// TIA Portal V16 export
// export: Created 2023-03-29T11:03:22.7150426Z, ExportSetting WithDefaults, DisplayName Totally Integrated Automation Portal, DisplayVersion V16 Update 6, DisplayName TIA Portal Version Control Interface, DisplayVersion V16 Update 2, DisplayName TIA Portal Openness, DisplayVersion V16 Update 6, DisplayName STEP 7 Professional, DisplayVersion V16 Update 6, DisplayName STEP 7 Safety, DisplayVersion V16, DisplayName WinCC Advanced, DisplayVersion V16 Update 6
FUNCTION_BLOCK "Startegia_sterowania"   // FB18, LAD
TITLE = Strategia przełączania
{ S7_Optimized_Access := 'TRUE' }
AUTHOR : rtecmer
VERSION : 0.1
// Funkcja przełącza stan aktywnego zbiornika w trybie napełniania i opróróżniana. Cykl pracy . Zbiornik opróżniany zostaje aktywny do napełniania a jeden pełny aktywny do przetłaczannia. 
// Znacznik blok_tank_x - blukuje zbiornik po zakonczonym cyklu do czasu aż wszystkie zbiorniki nie przejdą sekwencji.
// stored: AutoNumber true, IsIECCheckEnabled false, IsRetainMemResEnabled false, MemoryReserve 250, SetENOAutomatically false, UDAEnableTagReadback false
   VAR
      tmp_time_1 : Bool;   // pomocniczy bit do wyzwolenia opóźnionego resetu aktywnego zbiornika
      tmp_time_2 : Bool := false;   // pomocniczy bit do wyzwolenia opóźnionego resetu aktywnego zbiornika
      tmp_time_3 : Bool := false;   // pomocniczy bit do wyzwolenia opóźnionego resetu aktywnego zbiornika
      tmp_time_4 : Bool := false;   // pomocniczy bit do wyzwolenia opóźnionego resetu aktywnego zbiornika
   END_VAR
   VAR_TEMP   // added for the SCL form of the ladder/FBD networks
      _w1 : Bool;
      _w2 : Bool;
   END_VAR
BEGIN

REGION Network 2: jest zablokowany po pracy w sekwencji
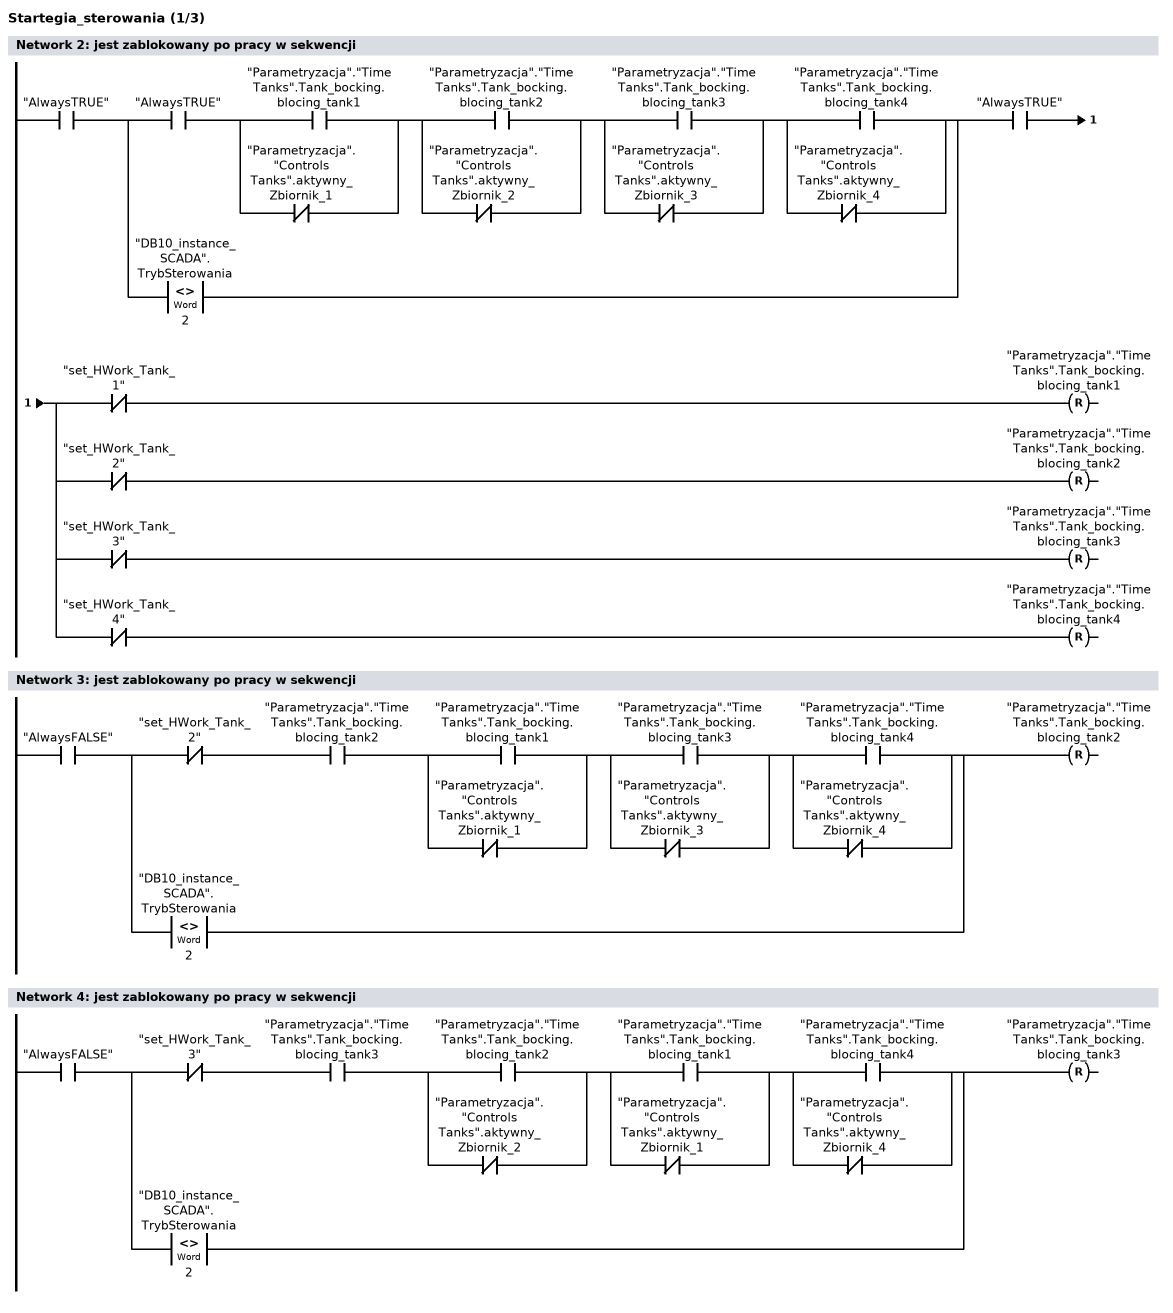
   RUNG wire#powerrail
      Contact( "AlwaysTRUE" )
      wire#w1
      Contact( "AlwaysTRUE" )
      wire#w2
      Contact( "Parametryzacja"."Time Tanks".Tank_bocking.blocing_tank1 )
      wire#w3
      Contact( "Parametryzacja"."Time Tanks".Tank_bocking.blocing_tank2 )
      wire#w4
      Contact( "Parametryzacja"."Time Tanks".Tank_bocking.blocing_tank3 )
      wire#w5
      Contact( "Parametryzacja"."Time Tanks".Tank_bocking.blocing_tank4 )
      wire#w6
      Contact( "AlwaysTRUE" )
      wire#w7
      I_Contact( "set_HWork_Tank_1" )
      R_Coil( "Parametryzacja"."Time Tanks".Tank_bocking.blocing_tank1 )
   END_RUNG
   RUNG wire#w2
      I_Contact( "Parametryzacja"."Controls Tanks".aktywny_Zbiornik_1 )
   END_RUNG wire#w3
   RUNG wire#w3
      I_Contact( "Parametryzacja"."Controls Tanks".aktywny_Zbiornik_2 )
   END_RUNG wire#w4
   RUNG wire#w4
      I_Contact( "Parametryzacja"."Controls Tanks".aktywny_Zbiornik_3 )
   END_RUNG wire#w5
   RUNG wire#w5
      I_Contact( "Parametryzacja"."Controls Tanks".aktywny_Zbiornik_4 )
   END_RUNG wire#w6
   RUNG wire#w1
      { S7_Templates := "SrcType := Word" } NE_Contact(in1 := "DB10_instance_SCADA".TrybSterowania, in2 := 2)
   END_RUNG wire#w6
   RUNG wire#w7
      I_Contact( "set_HWork_Tank_2" )
      R_Coil( "Parametryzacja"."Time Tanks".Tank_bocking.blocing_tank2 )
   END_RUNG
   RUNG wire#w7
      I_Contact( "set_HWork_Tank_3" )
      R_Coil( "Parametryzacja"."Time Tanks".Tank_bocking.blocing_tank3 )
   END_RUNG
   RUNG wire#w7
      I_Contact( "set_HWork_Tank_4" )
      R_Coil( "Parametryzacja"."Time Tanks".Tank_bocking.blocing_tank4 )
   END_RUNG
   // the same network as SCL:
   #_w1 := "AlwaysTRUE" AND (("AlwaysTRUE" AND ("Parametryzacja"."Time Tanks".Tank_bocking.blocing_tank1 OR NOT "Parametryzacja"."Controls Tanks".aktywny_Zbiornik_1) AND ("Parametryzacja"."Time Tanks".Tank_bocking.blocing_tank2 OR NOT "Parametryzacja"."Controls Tanks".aktywny_Zbiornik_2) AND ("Parametryzacja"."Time Tanks".Tank_bocking.blocing_tank3 OR NOT "Parametryzacja"."Controls Tanks".aktywny_Zbiornik_3) AND ("Parametryzacja"."Time Tanks".Tank_bocking.blocing_tank4 OR NOT "Parametryzacja"."Controls Tanks".aktywny_Zbiornik_4)) OR ("DB10_instance_SCADA".TrybSterowania <> 2)) AND "AlwaysTRUE";
   IF #_w1 AND NOT "set_HWork_Tank_1" THEN
       "Parametryzacja"."Time Tanks".Tank_bocking.blocing_tank1 := FALSE;
   END_IF;
   IF #_w1 AND NOT "set_HWork_Tank_2" THEN
       "Parametryzacja"."Time Tanks".Tank_bocking.blocing_tank2 := FALSE;
   END_IF;
   IF #_w1 AND NOT "set_HWork_Tank_3" THEN
       "Parametryzacja"."Time Tanks".Tank_bocking.blocing_tank3 := FALSE;
   END_IF;
   IF #_w1 AND NOT "set_HWork_Tank_4" THEN
       "Parametryzacja"."Time Tanks".Tank_bocking.blocing_tank4 := FALSE;
   END_IF;
END_REGION

REGION Network 3: jest zablokowany po pracy w sekwencji
   RUNG wire#powerrail
      Contact( "AlwaysFALSE" )
      wire#w1
      I_Contact( "set_HWork_Tank_2" )
      Contact( "Parametryzacja"."Time Tanks".Tank_bocking.blocing_tank2 )
      wire#w2
      Contact( "Parametryzacja"."Time Tanks".Tank_bocking.blocing_tank1 )
      wire#w3
      Contact( "Parametryzacja"."Time Tanks".Tank_bocking.blocing_tank3 )
      wire#w4
      Contact( "Parametryzacja"."Time Tanks".Tank_bocking.blocing_tank4 )
      wire#w5
      R_Coil( "Parametryzacja"."Time Tanks".Tank_bocking.blocing_tank2 )
   END_RUNG
   RUNG wire#w2
      I_Contact( "Parametryzacja"."Controls Tanks".aktywny_Zbiornik_1 )
   END_RUNG wire#w3
   RUNG wire#w3
      I_Contact( "Parametryzacja"."Controls Tanks".aktywny_Zbiornik_3 )
   END_RUNG wire#w4
   RUNG wire#w4
      I_Contact( "Parametryzacja"."Controls Tanks".aktywny_Zbiornik_4 )
   END_RUNG wire#w5
   RUNG wire#w1
      { S7_Templates := "SrcType := Word" } NE_Contact(in1 := "DB10_instance_SCADA".TrybSterowania, in2 := 2)
   END_RUNG wire#w5
   // the same network as SCL:
   IF "AlwaysFALSE" AND ((NOT "set_HWork_Tank_2" AND "Parametryzacja"."Time Tanks".Tank_bocking.blocing_tank2 AND ("Parametryzacja"."Time Tanks".Tank_bocking.blocing_tank1 OR NOT "Parametryzacja"."Controls Tanks".aktywny_Zbiornik_1) AND ("Parametryzacja"."Time Tanks".Tank_bocking.blocing_tank3 OR NOT "Parametryzacja"."Controls Tanks".aktywny_Zbiornik_3) AND ("Parametryzacja"."Time Tanks".Tank_bocking.blocing_tank4 OR NOT "Parametryzacja"."Controls Tanks".aktywny_Zbiornik_4)) OR ("DB10_instance_SCADA".TrybSterowania <> 2)) THEN
       "Parametryzacja"."Time Tanks".Tank_bocking.blocing_tank2 := FALSE;
   END_IF;
END_REGION

REGION Network 4: jest zablokowany po pracy w sekwencji
   RUNG wire#powerrail
      Contact( "AlwaysFALSE" )
      wire#w1
      I_Contact( "set_HWork_Tank_3" )
      Contact( "Parametryzacja"."Time Tanks".Tank_bocking.blocing_tank3 )
      wire#w2
      Contact( "Parametryzacja"."Time Tanks".Tank_bocking.blocing_tank2 )
      wire#w3
      Contact( "Parametryzacja"."Time Tanks".Tank_bocking.blocing_tank1 )
      wire#w4
      Contact( "Parametryzacja"."Time Tanks".Tank_bocking.blocing_tank4 )
      wire#w5
      R_Coil( "Parametryzacja"."Time Tanks".Tank_bocking.blocing_tank3 )
   END_RUNG
   RUNG wire#w2
      I_Contact( "Parametryzacja"."Controls Tanks".aktywny_Zbiornik_2 )
   END_RUNG wire#w3
   RUNG wire#w3
      I_Contact( "Parametryzacja"."Controls Tanks".aktywny_Zbiornik_1 )
   END_RUNG wire#w4
   RUNG wire#w4
      I_Contact( "Parametryzacja"."Controls Tanks".aktywny_Zbiornik_4 )
   END_RUNG wire#w5
   RUNG wire#w1
      { S7_Templates := "SrcType := Word" } NE_Contact(in1 := "DB10_instance_SCADA".TrybSterowania, in2 := 2)
   END_RUNG wire#w5
   // the same network as SCL:
   IF "AlwaysFALSE" AND ((NOT "set_HWork_Tank_3" AND "Parametryzacja"."Time Tanks".Tank_bocking.blocing_tank3 AND ("Parametryzacja"."Time Tanks".Tank_bocking.blocing_tank2 OR NOT "Parametryzacja"."Controls Tanks".aktywny_Zbiornik_2) AND ("Parametryzacja"."Time Tanks".Tank_bocking.blocing_tank1 OR NOT "Parametryzacja"."Controls Tanks".aktywny_Zbiornik_1) AND ("Parametryzacja"."Time Tanks".Tank_bocking.blocing_tank4 OR NOT "Parametryzacja"."Controls Tanks".aktywny_Zbiornik_4)) OR ("DB10_instance_SCADA".TrybSterowania <> 2)) THEN
       "Parametryzacja"."Time Tanks".Tank_bocking.blocing_tank3 := FALSE;
   END_IF;
END_REGION

REGION Network 5: Zbiornik 1 ustaw jako aktywny
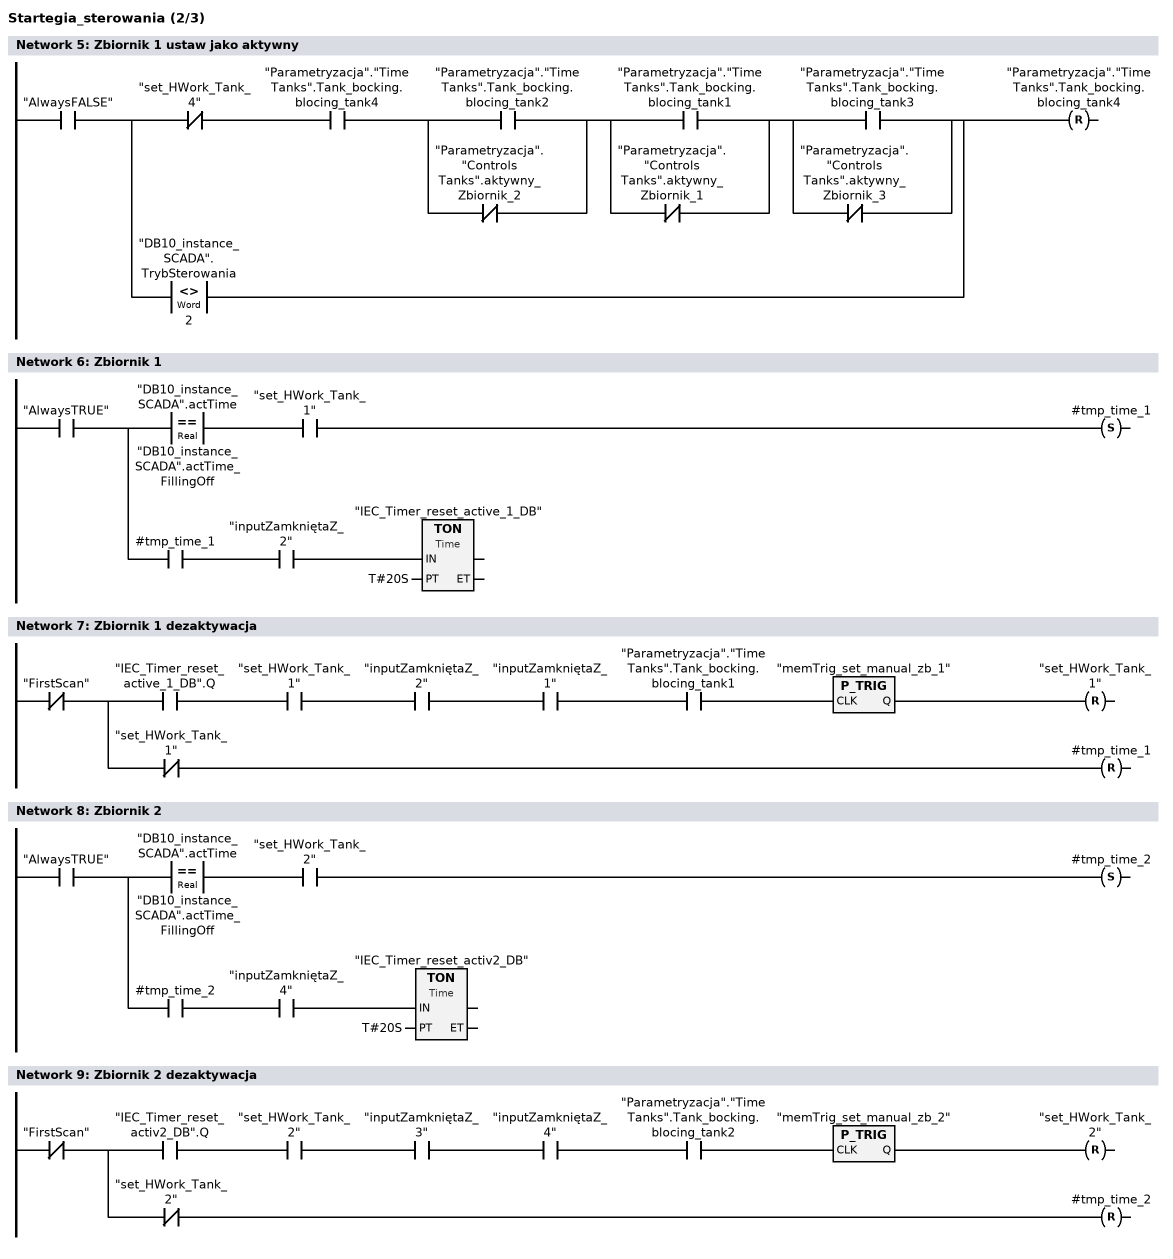
   RUNG wire#powerrail
      Contact( "AlwaysFALSE" )
      wire#w1
      I_Contact( "set_HWork_Tank_4" )
      Contact( "Parametryzacja"."Time Tanks".Tank_bocking.blocing_tank4 )
      wire#w2
      Contact( "Parametryzacja"."Time Tanks".Tank_bocking.blocing_tank2 )
      wire#w3
      Contact( "Parametryzacja"."Time Tanks".Tank_bocking.blocing_tank1 )
      wire#w4
      Contact( "Parametryzacja"."Time Tanks".Tank_bocking.blocing_tank3 )
      wire#w5
      R_Coil( "Parametryzacja"."Time Tanks".Tank_bocking.blocing_tank4 )
   END_RUNG
   RUNG wire#w2
      I_Contact( "Parametryzacja"."Controls Tanks".aktywny_Zbiornik_2 )
   END_RUNG wire#w3
   RUNG wire#w3
      I_Contact( "Parametryzacja"."Controls Tanks".aktywny_Zbiornik_1 )
   END_RUNG wire#w4
   RUNG wire#w4
      I_Contact( "Parametryzacja"."Controls Tanks".aktywny_Zbiornik_3 )
   END_RUNG wire#w5
   RUNG wire#w1
      { S7_Templates := "SrcType := Word" } NE_Contact(in1 := "DB10_instance_SCADA".TrybSterowania, in2 := 2)
   END_RUNG wire#w5
   // the same network as SCL:
   IF "AlwaysFALSE" AND ((NOT "set_HWork_Tank_4" AND "Parametryzacja"."Time Tanks".Tank_bocking.blocing_tank4 AND ("Parametryzacja"."Time Tanks".Tank_bocking.blocing_tank2 OR NOT "Parametryzacja"."Controls Tanks".aktywny_Zbiornik_2) AND ("Parametryzacja"."Time Tanks".Tank_bocking.blocing_tank1 OR NOT "Parametryzacja"."Controls Tanks".aktywny_Zbiornik_1) AND ("Parametryzacja"."Time Tanks".Tank_bocking.blocing_tank3 OR NOT "Parametryzacja"."Controls Tanks".aktywny_Zbiornik_3)) OR ("DB10_instance_SCADA".TrybSterowania <> 2)) THEN
       "Parametryzacja"."Time Tanks".Tank_bocking.blocing_tank4 := FALSE;
   END_IF;
END_REGION

REGION Network 6: Zbiornik 1
   RUNG wire#powerrail
      Contact( "AlwaysTRUE" )
      wire#w1
      { S7_Templates := "SrcType := Real" } EQ_Contact(in1 := "DB10_instance_SCADA".actTime, in2 := "DB10_instance_SCADA".actTime_FillingOff)
      Contact( "set_HWork_Tank_1" )
      S_Coil( #tmp_time_1 )
   END_RUNG
   RUNG wire#w1
      Contact( #tmp_time_1 )
      Contact( "inputZamkniętaZ_2" )
      { S7_Templates := "time_type := Time" } "IEC_Timer_reset_active_1_DB".TON(pt := T#20S, et =>)
   END_RUNG
   // the same network as SCL:
   IF "AlwaysTRUE" AND ("DB10_instance_SCADA".actTime = "DB10_instance_SCADA".actTime_FillingOff) AND "set_HWork_Tank_1" THEN
       #tmp_time_1 := TRUE;
   END_IF;
   "IEC_Timer_reset_active_1_DB".TON(IN := "AlwaysTRUE" AND #tmp_time_1 AND "inputZamkniętaZ_2", PT := T#20S);
END_REGION

REGION Network 7: Zbiornik 1 dezaktywacja
   RUNG wire#powerrail
      I_Contact( "FirstScan" )
      wire#w1
      Contact( "IEC_Timer_reset_active_1_DB".Q )
      Contact( "set_HWork_Tank_1" )
      Contact( "inputZamkniętaZ_2" )
      Contact( "inputZamkniętaZ_1" )
      Contact( "Parametryzacja"."Time Tanks".Tank_bocking.blocing_tank1 )
      P_Trig( "memTrig_set_manual_zb_1" )
      R_Coil( "set_HWork_Tank_1" )
   END_RUNG
   RUNG wire#w1
      I_Contact( "set_HWork_Tank_1" )
      R_Coil( #tmp_time_1 )
   END_RUNG
   // the same network as SCL:
   #_w1 := NOT "FirstScan" AND "IEC_Timer_reset_active_1_DB".Q AND "set_HWork_Tank_1" AND "inputZamkniętaZ_2" AND "inputZamkniętaZ_1" AND "Parametryzacja"."Time Tanks".Tank_bocking.blocing_tank1;
   #_w2 := #_w1 AND NOT "memTrig_set_manual_zb_1";   // rising edge
   "memTrig_set_manual_zb_1" := #_w1;
   IF #_w2 THEN "set_HWork_Tank_1" := FALSE; END_IF;
   IF NOT "FirstScan" AND NOT "set_HWork_Tank_1" THEN #tmp_time_1 := FALSE; END_IF;
END_REGION

REGION Network 8: Zbiornik 2
   RUNG wire#powerrail
      Contact( "AlwaysTRUE" )
      wire#w1
      { S7_Templates := "SrcType := Real" } EQ_Contact(in1 := "DB10_instance_SCADA".actTime, in2 := "DB10_instance_SCADA".actTime_FillingOff)
      Contact( "set_HWork_Tank_2" )
      S_Coil( #tmp_time_2 )
   END_RUNG
   RUNG wire#w1
      Contact( #tmp_time_2 )
      Contact( "inputZamkniętaZ_4" )
      { S7_Templates := "time_type := Time" } "IEC_Timer_reset_activ2_DB".TON(pt := T#20S, et =>)
   END_RUNG
   // the same network as SCL:
   IF "AlwaysTRUE" AND ("DB10_instance_SCADA".actTime = "DB10_instance_SCADA".actTime_FillingOff) AND "set_HWork_Tank_2" THEN
       #tmp_time_2 := TRUE;
   END_IF;
   "IEC_Timer_reset_activ2_DB".TON(IN := "AlwaysTRUE" AND #tmp_time_2 AND "inputZamkniętaZ_4", PT := T#20S);
END_REGION

REGION Network 9: Zbiornik 2 dezaktywacja
   RUNG wire#powerrail
      I_Contact( "FirstScan" )
      wire#w1
      Contact( "IEC_Timer_reset_activ2_DB".Q )
      Contact( "set_HWork_Tank_2" )
      Contact( "inputZamkniętaZ_3" )
      Contact( "inputZamkniętaZ_4" )
      Contact( "Parametryzacja"."Time Tanks".Tank_bocking.blocing_tank2 )
      P_Trig( "memTrig_set_manual_zb_2" )
      R_Coil( "set_HWork_Tank_2" )
   END_RUNG
   RUNG wire#w1
      I_Contact( "set_HWork_Tank_2" )
      R_Coil( #tmp_time_2 )
   END_RUNG
   // the same network as SCL:
   #_w1 := NOT "FirstScan" AND "IEC_Timer_reset_activ2_DB".Q AND "set_HWork_Tank_2" AND "inputZamkniętaZ_3" AND "inputZamkniętaZ_4" AND "Parametryzacja"."Time Tanks".Tank_bocking.blocing_tank2;
   #_w2 := #_w1 AND NOT "memTrig_set_manual_zb_2";   // rising edge
   "memTrig_set_manual_zb_2" := #_w1;
   IF #_w2 THEN "set_HWork_Tank_2" := FALSE; END_IF;
   IF NOT "FirstScan" AND NOT "set_HWork_Tank_2" THEN #tmp_time_2 := FALSE; END_IF;
END_REGION

REGION Network 10: Zbiornik 3
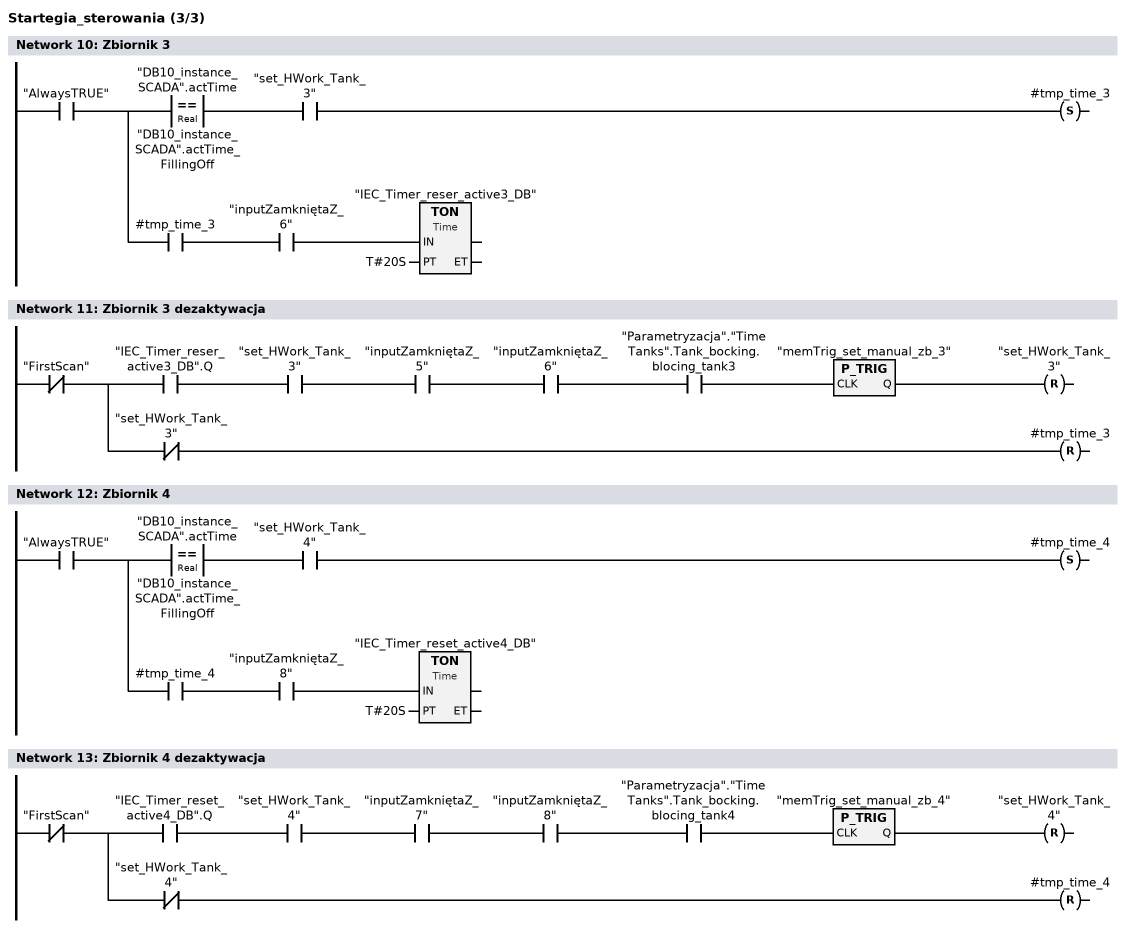
   RUNG wire#powerrail
      Contact( "AlwaysTRUE" )
      wire#w1
      { S7_Templates := "SrcType := Real" } EQ_Contact(in1 := "DB10_instance_SCADA".actTime, in2 := "DB10_instance_SCADA".actTime_FillingOff)
      Contact( "set_HWork_Tank_3" )
      S_Coil( #tmp_time_3 )
   END_RUNG
   RUNG wire#w1
      Contact( #tmp_time_3 )
      Contact( "inputZamkniętaZ_6" )
      { S7_Templates := "time_type := Time" } "IEC_Timer_reser_active3_DB".TON(pt := T#20S, et =>)
   END_RUNG
   // the same network as SCL:
   IF "AlwaysTRUE" AND ("DB10_instance_SCADA".actTime = "DB10_instance_SCADA".actTime_FillingOff) AND "set_HWork_Tank_3" THEN
       #tmp_time_3 := TRUE;
   END_IF;
   "IEC_Timer_reser_active3_DB".TON(IN := "AlwaysTRUE" AND #tmp_time_3 AND "inputZamkniętaZ_6", PT := T#20S);
END_REGION

REGION Network 11: Zbiornik 3 dezaktywacja
   RUNG wire#powerrail
      I_Contact( "FirstScan" )
      wire#w1
      Contact( "IEC_Timer_reser_active3_DB".Q )
      Contact( "set_HWork_Tank_3" )
      Contact( "inputZamkniętaZ_5" )
      Contact( "inputZamkniętaZ_6" )
      Contact( "Parametryzacja"."Time Tanks".Tank_bocking.blocing_tank3 )
      P_Trig( "memTrig_set_manual_zb_3" )
      R_Coil( "set_HWork_Tank_3" )
   END_RUNG
   RUNG wire#w1
      I_Contact( "set_HWork_Tank_3" )
      R_Coil( #tmp_time_3 )
   END_RUNG
   // the same network as SCL:
   #_w1 := NOT "FirstScan" AND "IEC_Timer_reser_active3_DB".Q AND "set_HWork_Tank_3" AND "inputZamkniętaZ_5" AND "inputZamkniętaZ_6" AND "Parametryzacja"."Time Tanks".Tank_bocking.blocing_tank3;
   #_w2 := #_w1 AND NOT "memTrig_set_manual_zb_3";   // rising edge
   "memTrig_set_manual_zb_3" := #_w1;
   IF #_w2 THEN "set_HWork_Tank_3" := FALSE; END_IF;
   IF NOT "FirstScan" AND NOT "set_HWork_Tank_3" THEN #tmp_time_3 := FALSE; END_IF;
END_REGION

REGION Network 12: Zbiornik 4
   RUNG wire#powerrail
      Contact( "AlwaysTRUE" )
      wire#w1
      { S7_Templates := "SrcType := Real" } EQ_Contact(in1 := "DB10_instance_SCADA".actTime, in2 := "DB10_instance_SCADA".actTime_FillingOff)
      Contact( "set_HWork_Tank_4" )
      S_Coil( #tmp_time_4 )
   END_RUNG
   RUNG wire#w1
      Contact( #tmp_time_4 )
      Contact( "inputZamkniętaZ_8" )
      { S7_Templates := "time_type := Time" } "IEC_Timer_reset_active4_DB".TON(pt := T#20S, et =>)
   END_RUNG
   // the same network as SCL:
   IF "AlwaysTRUE" AND ("DB10_instance_SCADA".actTime = "DB10_instance_SCADA".actTime_FillingOff) AND "set_HWork_Tank_4" THEN
       #tmp_time_4 := TRUE;
   END_IF;
   "IEC_Timer_reset_active4_DB".TON(IN := "AlwaysTRUE" AND #tmp_time_4 AND "inputZamkniętaZ_8", PT := T#20S);
END_REGION

REGION Network 13: Zbiornik 4 dezaktywacja
   RUNG wire#powerrail
      I_Contact( "FirstScan" )
      wire#w1
      Contact( "IEC_Timer_reset_active4_DB".Q )
      Contact( "set_HWork_Tank_4" )
      Contact( "inputZamkniętaZ_7" )
      Contact( "inputZamkniętaZ_8" )
      Contact( "Parametryzacja"."Time Tanks".Tank_bocking.blocing_tank4 )
      P_Trig( "memTrig_set_manual_zb_4" )
      R_Coil( "set_HWork_Tank_4" )
   END_RUNG
   RUNG wire#w1
      I_Contact( "set_HWork_Tank_4" )
      R_Coil( #tmp_time_4 )
   END_RUNG
   // the same network as SCL:
   #_w1 := NOT "FirstScan" AND "IEC_Timer_reset_active4_DB".Q AND "set_HWork_Tank_4" AND "inputZamkniętaZ_7" AND "inputZamkniętaZ_8" AND "Parametryzacja"."Time Tanks".Tank_bocking.blocing_tank4;
   #_w2 := #_w1 AND NOT "memTrig_set_manual_zb_4";   // rising edge
   "memTrig_set_manual_zb_4" := #_w1;
   IF #_w2 THEN "set_HWork_Tank_4" := FALSE; END_IF;
   IF NOT "FirstScan" AND NOT "set_HWork_Tank_4" THEN #tmp_time_4 := FALSE; END_IF;
END_REGION
END_FUNCTION_BLOCK
